Fanuc KAREL source: ko00090.KL

-- PROVISIONAL review KL for V770-1; original PC SHA256 f961c115538f44961477265ff3d61782cc044354459a72f4379cfce20f355d0b
-- Incomplete behavior may be omitted. Consult companion uncertainty JSON. Do not deploy.
PROGRAM KO00090
%NOLOCKGROUP
BEGIN
  -- UNRESOLVED_PC offsets 5-12; opcodes 9D,23
  -- UNRESOLVED_PC offsets 17-69; opcodes 27,27,49,7E,AD,27,49,7E,AD,22,31,7E,4A
  -- UNRESOLVED_PC offsets 74-78; opcodes 7F
END KO00090
